// TIA Portal V18 export
// export: Created 2025-12-01T17:52:52.2638005Z, ExportSetting None, DisplayName Totally Integrated Automation Portal, DisplayVersion V18 Update 5, DisplayName TIA Portal Openness, DisplayVersion V18 Update 5, DisplayName TIA Portal Teamcenter Gateway, DisplayVersion V18, DisplayName TIA Portal Version Control Interface, DisplayVersion V18, DisplayName STEP 7 Professional, DisplayVersion V18 Update 5, DisplayName STEP 7 Safety, DisplayVersion V18, DisplayName WinCC Professional, DisplayVersion V18 Update 5
Screen "9900Cylinder"  1280x800, Number=12, Template=T1
  ScreenLayer 
    Rectangle "矩形_1" at 28,89 size 45x100
    Rectangle "矩形_2" at 28,89 size 45x50
    Polygon "多边形_1" at 135,93 size 35x100
    Polygon "多边形_2" at 91,93 size 35x100
      RangeAppearanceAnimation "RangeAppearanceAnimation"
        tag 
        0..0: back #ff0000, fore #181c31
        1..1: back #d9d9d9, fore #181c31
  ScreenLayer 
    GraphicIOField "geaInitialPosition" at 203,93 size 136x82  Mode=Output, PictureList=HomeStatus
      RangeAppearanceAnimation "RangeAppearanceAnimation"
        tag 
        0..0: back #647887, fore #647887
        1..1: back #5dd746, fore #647887
      ProcessValue := ST_AutoStatus
